{attribute 'qualified_only'}
{attribute 'strict'}
TYPE eLEDMode :
(
	On,
	Dimmed,
	SlowFlashing,
	FastFlashing
);
END_TYPE

(* stored: Version 1.1.0.1, ProductVersion 3.1.4024.12
   DUT eLEDMode: Id {ccc2dfe6-c924-4e60-8375-fc91686a2ce4} *)
